(* IEC 61131-3 sources: rules_plc/examples/direct_address, 2 files *)

(* ---- lib.st ---- *)
(*
Example library: defines a FUNCTION_BLOCK `Incrementer` that stores a
counter and places an integer at a direct address. This demonstrates
an st_library providing a reusable function block.
*)

FUNCTION_BLOCK Incrementer
    VAR
        Counter : INT := 0;
        Addr AT %QX0.0.1.0 : INT; (* direct address example *)
    END_VAR
    Counter := Counter + 1;
END_FUNCTION_BLOCK

(* ---- direct_address.st ---- *)
(*
Example program: instantiates `Incrementer` from the library, increments
its counter, and stores the result in a local variable. This file is the
`PROGRAM` entrypoint used by `st_binary`.
*)

PROGRAM direct_address
    VAR
        fb : Incrementer;
        out : INT;
    END_VAR
    fb();
END_PROGRAM
